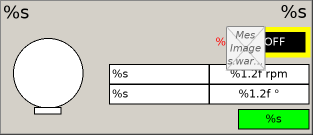
VISUALIZATION VISU_AXE_STD1_ROT_ABS_OSC  // 313x135
VAR_IN_OUT
	m_Input_MOTEUR: BLOCK_AXE_STD1_OSCILLANT;
	m_Input_PRG_MOUVEMENT_PS: BLOCK_PRG_MOUVEMENT_PS;
END_VAR
VAR_Input
	m_Input_ID_NOM_XML : INT;
	m_Input_INDEX_MOTEUR : INT;
	m_Input_Ref_Trf:	INT;
	m_Input_NumFrame_Manu:	USINT;		(*numéro de frame à afficher dans le synoptique MANUEL*)
END_VAR
    Rectangle (0,0 313x135), "%s", text list: 'TextList_Type_Moteur', text index: m_Input_ID_NOM_XML
    Rectangle (223,4 87x16), "%s", text variable: m_Input_MOTEUR.MNEMO
    RoundedRectangle (109,64 100x20), "%s", text list: 'TextList_Moteurs', text index: 7
    RoundedRectangle (109,84 100x20), "%s", text list: 'TextList_Moteurs', text index: 9
    RoundedRectangle (209,64 100x20), "%1.2f rpm", text variable: m_Input_MOTEUR.STATE_Vit
    RoundedRectangle (209,84 100x20), "%1.2f °", text variable: m_Input_MOTEUR.STATE_Pos
    RoundedRectangle (238,109 71x20), "%s", invisible if: m_Input_MOTEUR.STATE_Homed OR m_Input_MOTEUR.CONF_No_Ref, text list: 'TextList_Moteurs', text index: 11
    RoundedRectangle (238,109 71x20), "%s", invisible if: NOT m_Input_MOTEUR.STATE_Homed OR m_Input_MOTEUR.CONF_No_Ref, text list: 'TextList_Moteurs', text index: 11
    RoundedRectangle (240,27 70x30), invisible if: NOT m_Input_MOTEUR.OP_Validation.OK
    RoundedRectangle (240,27 70x30), invisible if: NOT m_Input_MOTEUR.OP_Validation.AR
    RoundedRectangle (240,27 70x30), invisible if: NOT m_Input_MOTEUR.OP_Validation.EC
    RoundedRectangle (245,32 60x20), "ON", invisible if: m_Input_MOTEUR.STATE_Ar
    RoundedRectangle (245,32 60x20), "OFF", invisible if: NOT m_Input_MOTEUR.STATE_Ar
    Rectangle (165,34 67x21), "%i", text variable: m_Input_MOTEUR.STATE_Err, invisible if: NOT m_Input_MOTEUR.STATE_NOK
    Image (226,26 39x44), invisible if: NOT m_Input_MOTEUR.STATE_NOK, image: MesImages.warning
    Rectangle (0,0 313x135)
        OnMouseClick: execute { .VISU_INDEX_MANU := m_Input_NumFrame_Manu; }
        OnMouseClick: change screen: SYN_MANUEL
    Ellipse (13,38 70x70)
    Rectangle (34,107 27x7)
END_VISUALIZATION

(* stored: Version 1.1.0.1, ProductVersion 3.1.4024.10
   Visu VISU_AXE_STD1_ROT_ABS_OSC: Id {26b01457-8731-408d-a777-6d479604182e} *)
